INTERFACE PUBLIC UnsuspendingCommands

METHOD PUBLIC Abort
END_METHOD

METHOD PUBLIC StateComplete
END_METHOD

METHOD PUBLIC Stop
END_METHOD

END_INTERFACE

(* stored: Version 1.1.0.1, ProductVersion 3.1.4026.12
   Itf UnsuspendingCommands: Id {100e6468-f259-0ece-08ab-ed447511f482}
   Method Abort: Id {4b414512-4c8f-41e4-bd5c-cf0e27928011}
   Method StateComplete: Id {6b7bf8ad-dd2f-4358-9f09-fdfa46e48b59}
   Method Stop: Id {d2e2d137-0f37-43c9-b678-bba7b4ffe537} *)
